{attribute 'qualified_only'}
{attribute 'TcHmiSymbol.AddSymbol'}
VAR_GLOBAL
    stRobot : ST_HmiRobot := (Name := 'Robot');

    // Robot tuning parameters, request flags, and the STATE/CMD channel --
    // all exchanged over TCP:6001 by FB_RobotTcpClient, which is the SOLE
    // robot channel (the discrete-I/O handshake was retired 2026-07-26).
    // The 11 tuning params are read/write: editing one here is detected by
    // the FB's shadow-copy comparison and pushed to the robot.
    stParams : ST_RobotParams;

    // TCP client target. PLC dials the robot's server. Host is set by the
    // commissioner (robot IP, e.g. '192.168.201.1'); port matches global.lua.
    sRobotHost : STRING := '192.168.201.1';
    nRobotPort : UINT := 6001;

    // Master enable for the TCP client. FALSE holds it disconnected.
    bTcpEnable : BOOL := TRUE;
END_VAR

(* stored: Version 1.1.0.1, ProductVersion 3.1.4026.18
   GVL GVL_Robot: Id {2f2957ad-9ce7-4061-8c32-dda5963bc0f5} *)
